Yaskawa INFORM job: CIRCULAR_S3.JBI

/JOB
//NAME CIRCULAR_S3
//POS
///NPOS 74,74,74,0,0,0
///TOOL 2
///POSTYPE PULSE
///PULSE
C00000=-121165,-3775,-12390,38142,6344,60040
C00001=-121367,-3602,-27967,39582,13719,57509
C00002=-121392,-319,-28319,39973,15020,57032
C00003=-121402,1038,-28413,40140,15532,56841
C00004=-121437,4653,-25587,39723,14109,56135
C00005=-121505,10655,-20712,38689,11227,54750
C00006=-121532,14229,-17726,38083,9745,54071
C00007=-121562,16831,-15495,37431,8291,53384
C00008=-121610,23055,-10032,35972,5322,52028
C00009=-121651,29298,-4349,34323,2318,50665
C00010=-121685,35546,1541,32496,-705,49284
C00011=-121714,41725,7563,30506,-3716,47879
C00012=-121738,47856,13725,28344,-6712,46431
C00013=-121760,53887,19962,26006,-9666,44924
C00014=-121780,59801,26245,23483,-12549,43350
C00015=-121799,65536,32489,20764,-15325,41693
C00016=-121819,71090,38673,17815,-17969,39931
C00017=-121839,76359,44658,14629,-20415,38059
C00018=-121860,81284,50355,11190,-22612,36066
C00019=-121882,85724,55567,7499,-24476,33949
C00020=-121903,89548,60111,3571,-25927,31713
C00021=-121922,92529,63680,-525,-26855,29386
C00022=-121935,94470,66007,-4673,-27173,27023
C00023=-121936,95184,66837,-8774,-26812,24663
C00024=-121922,94612,66095,-12680,-25771,22377
C00025=-121888,92807,63855,-16310,-24096,20200
C00026=-121834,89952,60365,-19611,-21893,18163
C00027=-121757,86278,55938,-22567,-19288,16279
C00028=-121660,81965,50820,-25222,-16375,14527
C00029=-121542,77175,45233,-27611,-13238,12891
C00030=-121405,72028,39340,-29766,-9949,11357
C00031=-121250,66621,33277,-31718,-6560,9904
C00032=-121076,60982,27094,-33502,-3091,8509
C00033=-120886,55192,20897,-35123,411,7161
C00034=-120678,49267,14719,-36590,3931,5842
C00035=-120455,43255,8623,-37902,7443,4536
C00036=-120216,37156,2621,-39052,10942,3227
C00037=-119964,31023,-3225,-40017,14402,1901
C00038=-119701,24886,-8883,-40769,17795,549
C00039=-119428,18749,-14344,-41279,21133,-857
C00040=-119149,12639,-19586,-41500,24390,-2332
C00041=-118867,6587,-24585,-41378,27563,-3901
C00042=-118588,611,-29330,-40850,30627,-5586
C00043=-118320,-5205,-33770,-39849,33545,-7400
C00044=-118069,-10866,-37924,-38298,36304,-9377
C00045=-117847,-16304,-41759,-36123,38870,-11540
C00046=-117665,-21485,-45275,-33262,41198,-13908
C00047=-117535,-26338,-48445,-29674,43245,-16492
C00048=-117467,-30845,-51284,-25333,44973,-19310
C00049=-117472,-34918,-53756,-20302,46330,-22333
C00050=-117552,-38524,-55865,-14691,47281,-25527
C00051=-117704,-41588,-57588,-8683,47804,-28830
C00052=-117917,-44079,-58930,-2489,47896,-32179
C00053=-118175,-45935,-59877,3647,47576,-35491
C00054=-118459,-47133,-60441,9500,46881,-38689
C00055=-118758,-47644,-60623,14968,45853,-41756
C00056=-119056,-47464,-60433,19936,44539,-44656
C00057=-119348,-46585,-59873,24377,42977,-47392
C00058=-119627,-45023,-58947,28263,41207,-49960
C00059=-119888,-42814,-57665,31582,39270,-52357
C00060=-120129,-39986,-56023,34367,37183,-54605
C00061=-120351,-36588,-54025,36639,34968,-56716
C00062=-120551,-32672,-51673,38419,32646,-58698
C00063=-120731,-28308,-48975,39738,30232,-60562
C00064=-120891,-23520,-45918,40630,27722,-62329
C00065=-121033,-18396,-42523,41122,25135,-64004
C00066=-121097,-15903,-40821,41224,23807,-64808
C00067=-121157,-12971,-38786,41246,22476,-65599
C00068=-121264,-7315,-34729,41034,19751,-67124
C00069=-121358,-1448,-30342,40516,16958,-68596
C00070=-121402,1038,-28413,40140,15532,-69314
C00071=-121392,-319,-28319,39973,15020,-69124
C00072=-121367,-3602,-27967,39582,13719,-68646
C00073=-121165,-3775,-12390,38142,6344,-66116
///TOOL 0
BC00000=204858
BC00001=204858
BC00002=200997
BC00003=199452
BC00004=200722
BC00005=201987
BC00006=202594
BC00007=202710
BC00008=202840
BC00009=202368
BC00010=201301
BC00011=199655
BC00012=197441
BC00013=194683
BC00014=191409
BC00015=187660
BC00016=183447
BC00017=178833
BC00018=173846
BC00019=168548
BC00020=162964
BC00021=157174
BC00022=151240
BC00023=145200
BC00024=139113
BC00025=133037
BC00026=127021
BC00027=121167
BC00028=115490
BC00029=110067
BC00030=104939
BC00031=100172
BC00032=95776
BC00033=91825
BC00034=88336
BC00035=85359
BC00036=82906
BC00037=81018
BC00038=79705
BC00039=78982
BC00040=78852
BC00041=79323
BC00042=80391
BC00043=82036
BC00044=84251
BC00045=87008
BC00046=90283
BC00047=94031
BC00048=98244
BC00049=102858
BC00050=107845
BC00051=113144
BC00052=118727
BC00053=124517
BC00054=130451
BC00055=136491
BC00056=142579
BC00057=148654
BC00058=154671
BC00059=160524
BC00060=166201
BC00061=171624
BC00062=176753
BC00063=181519
BC00064=185915
BC00065=189866
BC00066=191442
BC00067=193355
BC00068=196332
BC00069=198785
BC00070=199452
BC00071=200997
BC00072=204858
BC00073=204858
EC00000=-379617,176269
EC00001=-379617,176269
EC00002=-379617,176269
EC00003=-379617,176269
EC00004=-379617,176269
EC00005=-379617,176269
EC00006=-379617,176269
EC00007=-379617,176269
EC00008=-379617,176269
EC00009=-379617,176269
EC00010=-379617,176269
EC00011=-379617,176269
EC00012=-379617,176269
EC00013=-379617,176269
EC00014=-379617,176269
EC00015=-379617,176269
EC00016=-379617,176269
EC00017=-379617,176269
EC00018=-379617,176269
EC00019=-379617,176269
EC00020=-379617,176269
EC00021=-379617,176269
EC00022=-379617,176269
EC00023=-379617,176269
EC00024=-379617,176269
EC00025=-379617,176269
EC00026=-379617,176269
EC00027=-379617,176269
EC00028=-379617,176269
EC00029=-379617,176269
EC00030=-379617,176269
EC00031=-379617,176269
EC00032=-379617,176269
EC00033=-379617,176269
EC00034=-379617,176269
EC00035=-379617,176269
EC00036=-379617,176269
EC00037=-379617,176269
EC00038=-379617,176269
EC00039=-379617,176269
EC00040=-379617,176269
EC00041=-379617,176269
EC00042=-379617,176269
EC00043=-379617,176269
EC00044=-379617,176269
EC00045=-379617,176269
EC00046=-379617,176269
EC00047=-379617,176269
EC00048=-379617,176269
EC00049=-379617,176269
EC00050=-379617,176269
EC00051=-379617,176269
EC00052=-379617,176269
EC00053=-379617,176269
EC00054=-379617,176269
EC00055=-379617,176269
EC00056=-379617,176269
EC00057=-379617,176269
EC00058=-379617,176269
EC00059=-379617,176269
EC00060=-379617,176269
EC00061=-379617,176269
EC00062=-379617,176269
EC00063=-379617,176269
EC00064=-379617,176269
EC00065=-379617,176269
EC00066=-379617,176269
EC00067=-379617,176269
EC00068=-379617,176269
EC00069=-379617,176269
EC00070=-379617,176269
EC00071=-379617,176269
EC00072=-379617,176269
EC00073=-379617,176269
//INST
///DATE 2026/05/13 10:02
///ATTR SC,RW
///GROUP1 RB1,BS1
///GROUP2 ST1
NOP
'Circular_s3
MEMOF
CLEAR MPF
'Path W3
SSFTOF
MOVJ C00000 BC00000 VJ=100.00  +MOVJ EC00000 VJ=100.00
SMOVL C00001 BC00001 V=1000.0  +MOVJ EC00001
SMOVL C00002 BC00002 V=400.0  +MOVJ EC00002
SMOVL C00003 BC00003 V=10.0 PL=0  +MOVJ EC00003
SMOVL C00004 BC00004 V=10.0  +MOVJ EC00004
SMOVL C00005 BC00005 V=10.0  +MOVJ EC00005
SMOVL C00006 BC00006 V=10.0  +MOVJ EC00006
SMOVL C00007 BC00007 V=10.0  +MOVJ EC00007
SMOVL C00008 BC00008 V=10.0  +MOVJ EC00008
SMOVL C00009 BC00009 V=10.0  +MOVJ EC00009
SMOVL C00010 BC00010 V=10.0  +MOVJ EC00010
SMOVL C00011 BC00011 V=10.0  +MOVJ EC00011
SMOVL C00012 BC00012 V=10.0  +MOVJ EC00012
SMOVL C00013 BC00013 V=10.0  +MOVJ EC00013
SMOVL C00014 BC00014 V=10.0  +MOVJ EC00014
SMOVL C00015 BC00015 V=10.0  +MOVJ EC00015
SMOVL C00016 BC00016 V=10.0  +MOVJ EC00016
SMOVL C00017 BC00017 V=10.0  +MOVJ EC00017
SMOVL C00018 BC00018 V=10.0  +MOVJ EC00018
SMOVL C00019 BC00019 V=10.0  +MOVJ EC00019
SMOVL C00020 BC00020 V=10.0  +MOVJ EC00020
SMOVL C00021 BC00021 V=10.0  +MOVJ EC00021
SMOVL C00022 BC00022 V=10.0  +MOVJ EC00022
SMOVL C00023 BC00023 V=10.0  +MOVJ EC00023
SMOVL C00024 BC00024 V=10.0  +MOVJ EC00024
SMOVL C00025 BC00025 V=10.0  +MOVJ EC00025
SMOVL C00026 BC00026 V=10.0  +MOVJ EC00026
SMOVL C00027 BC00027 V=10.0  +MOVJ EC00027
SMOVL C00028 BC00028 V=10.0  +MOVJ EC00028
SMOVL C00029 BC00029 V=10.0  +MOVJ EC00029
SMOVL C00030 BC00030 V=10.0  +MOVJ EC00030
SMOVL C00031 BC00031 V=10.0  +MOVJ EC00031
SMOVL C00032 BC00032 V=10.0  +MOVJ EC00032
SMOVL C00033 BC00033 V=10.0  +MOVJ EC00033
SMOVL C00034 BC00034 V=10.0  +MOVJ EC00034
SMOVL C00035 BC00035 V=10.0  +MOVJ EC00035
SMOVL C00036 BC00036 V=10.0  +MOVJ EC00036
SMOVL C00037 BC00037 V=10.0  +MOVJ EC00037
SMOVL C00038 BC00038 V=10.0  +MOVJ EC00038
SMOVL C00039 BC00039 V=10.0  +MOVJ EC00039
SMOVL C00040 BC00040 V=10.0  +MOVJ EC00040
SMOVL C00041 BC00041 V=10.0  +MOVJ EC00041
SMOVL C00042 BC00042 V=10.0  +MOVJ EC00042
SMOVL C00043 BC00043 V=10.0  +MOVJ EC00043
SMOVL C00044 BC00044 V=10.0  +MOVJ EC00044
SMOVL C00045 BC00045 V=10.0  +MOVJ EC00045
SMOVL C00046 BC00046 V=10.0  +MOVJ EC00046
SMOVL C00047 BC00047 V=10.0  +MOVJ EC00047
SMOVL C00048 BC00048 V=10.0  +MOVJ EC00048
SMOVL C00049 BC00049 V=10.0  +MOVJ EC00049
SMOVL C00050 BC00050 V=10.0  +MOVJ EC00050
SMOVL C00051 BC00051 V=10.0  +MOVJ EC00051
SMOVL C00052 BC00052 V=10.0  +MOVJ EC00052
SMOVL C00053 BC00053 V=10.0  +MOVJ EC00053
SMOVL C00054 BC00054 V=10.0  +MOVJ EC00054
SMOVL C00055 BC00055 V=10.0  +MOVJ EC00055
SMOVL C00056 BC00056 V=10.0  +MOVJ EC00056
SMOVL C00057 BC00057 V=10.0  +MOVJ EC00057
SMOVL C00058 BC00058 V=10.0  +MOVJ EC00058
SMOVL C00059 BC00059 V=10.0  +MOVJ EC00059
SMOVL C00060 BC00060 V=10.0  +MOVJ EC00060
SMOVL C00061 BC00061 V=10.0  +MOVJ EC00061
SMOVL C00062 BC00062 V=10.0  +MOVJ EC00062
SMOVL C00063 BC00063 V=10.0  +MOVJ EC00063
SMOVL C00064 BC00064 V=10.0  +MOVJ EC00064
SMOVL C00065 BC00065 V=10.0  +MOVJ EC00065
SMOVL C00066 BC00066 V=10.0  +MOVJ EC00066
SMOVL C00067 BC00067 V=10.0  +MOVJ EC00067
SMOVL C00068 BC00068 V=10.0  +MOVJ EC00068
SMOVL C00069 BC00069 V=10.0  +MOVJ EC00069
SMOVL C00070 BC00070 V=10.0  +MOVJ EC00070
SMOVL C00071 BC00071 V=400.0  +MOVJ EC00071
SMOVL C00072 BC00072 V=1000.0  +MOVJ EC00072
SMOVL C00073 BC00073 V=1000.0  +MOVJ EC00073
'EndPath W3
END
